FUNCTION_BLOCK SkillToLoad (* Basic Function Block Type *)
  (* Standard: 61499-2 *)
  (* Version 0.0, 9/24/2024, midxav, Template *)
  PACKAGE Main;
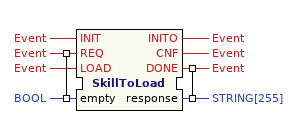
  EVENT_INPUT
    INIT; (* Initialization Request *)
    REQ WITH empty;
    LOAD;
  END_EVENT
  EVENT_OUTPUT
    INITO; (* Initialization Confirm *)
    CNF; (* Execution Confirmation *)
    DONE WITH response;
  END_EVENT
  VAR_INPUT
    empty : BOOL;
  END_VAR
  VAR_OUTPUT
    response : STRING[255];
  END_VAR
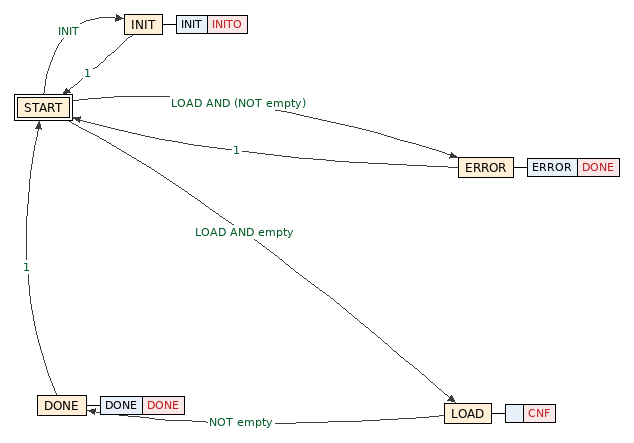
  EC_STATES
    START; (* Initial State *)
    INIT : INIT -> INITO; (* Initialization *)
    LOAD : -> CNF; (* Normal execution *)
    DONE : DONE -> DONE;
    ERROR : ERROR -> DONE;
  END_STATES
  EC_TRANSITIONS
    START TO INIT := INIT;
    INIT TO START := 1;
    START TO LOAD := LOAD AND empty;
    LOAD TO DONE := NOT empty;
    DONE TO START := 1;
    START TO ERROR := LOAD AND (NOT empty);
    ERROR TO START := 1;
  END_TRANSITIONS
  ALGORITHM INIT IN ST: (* Initialization algorithm *)
;
  END_ALGORITHM
  ALGORITHM DONE IN ST: (* Normally executed algorithm *)
response:='LOADED WP';
  END_ALGORITHM
  ALGORITHM ERROR IN ST:
response:='MAG NOT EMPTY';
  END_ALGORITHM
END_FUNCTION_BLOCK
